screen "performance_1" 1024x761
   IOField "I/O field_73" at 11,174 size 59x47; FormatPattern 99.99
      ProcessValue <- "Suction_press"
   IOField "I/O field_74" at 68,174 size 59x47; FormatPattern 99.99
      ProcessValue <- "Discharge_Press"
   IOField "I/O field_75" at 126,174 size 59x47; FormatPattern 99.99
      ProcessValue <- "Tag_9"
   IOField "I/O field_76" at 185,174 size 59x47; FormatPattern 99.99
      ProcessValue <- "P4"
   IOField "I/O field_77" at 241,174 size 59x47; FormatPattern 99.99
      ProcessValue <- "Torque"
   IOField "I/O field_78" at 299,174 size 59x47; FormatPattern 9999
      ProcessValue <- "RPM"
   IOField "I/O field_79" at 356,174 size 59x47; FormatPattern 99.99
      ProcessValue <- "Tag_33"
   IOField "I/O field_80" at 413,174 size 59x47; FormatPattern 99.99
      ProcessValue <- "VS"
   IOField "I/O field_81" at 470,174 size 59x47; FormatPattern 99.99
      ProcessValue <- "Vd"
   IOField "I/O field_82" at 527,174 size 59x47; FormatPattern 99.99
      ProcessValue <- "Q"
   IOField "I/O field_83" at 586,171 size 59x47; FormatPattern 99.99
      ProcessValue <- "H"
   IOField "I/O field_84" at 642,174 size 59x47; FormatPattern 9999.99
      ProcessValue <- "Shaft_power"
   IOField "I/O field_1" at 700,175 size 59x47; FormatPattern 99.99
      ProcessValue <- "QARS"
   IOField "I/O field_2" at 756,176 size 59x47; FormatPattern 99.99
      ProcessValue <- "H_ARS"
   IOField "I/O field_3" at 813,176 size 59x47; FormatPattern 9999.9
      ProcessValue <- "SP_ARS"
   IOField "I/O field_4" at 870,176 size 59x47; FormatPattern 99.99
      ProcessValue <- "Efficiency"
   IOField "I/O field_5" at 927,178 size 59x47; FormatPattern 99.9
      ProcessValue <- "Npsh"
   IOField "I/O field_6" at 11,220 size 59x47; FormatPattern 99.99
      ProcessValue <- "P1P2_Pressurep1p2{0}"
   IOField "I/O field_7" at 68,220 size 59x47; FormatPattern 99.99
      ProcessValue <- "P1P2_Pressurep1p2{6}"
   IOField "I/O field_8" at 126,220 size 59x47; FormatPattern 99.99
      ProcessValue <- "P3P4_Pressure34{0}"
   IOField "I/O field_9" at 185,220 size 59x47; FormatPattern 99.99
      ProcessValue <- "P3P4_Pressure34{6}"
   IOField "I/O field_10" at 241,220 size 59x47; FormatPattern 99.99
      ProcessValue <- "TS_TS{0}"
   IOField "I/O field_11" at 298,220 size 59x47; FormatPattern 9999
      ProcessValue <- "TS_TS{6}"
   IOField "I/O field_12" at 355,220 size 59x47; FormatPattern 99.99
      ProcessValue <- "Vib_vibration{0}"
   IOField "I/O field_13" at 412,220 size 59x47; FormatPattern 99.99
      ProcessValue <- "VSVD_VsVd{0}"
   IOField "I/O field_14" at 469,220 size 59x47; FormatPattern 99.99
      ProcessValue <- "VSVD_VsVd{6}"
   IOField "I/O field_15" at 527,220 size 59x47; FormatPattern 99.99
      ProcessValue <- "QH_QH{0}"
   IOField "I/O field_16" at 584,220 size 59x47; FormatPattern 99.99
      ProcessValue <- "QH_QH{6}"
   IOField "I/O field_17" at 642,220 size 59x47; FormatPattern 9999.99
      ProcessValue <- "shftP.Pars_shaftP{0}"
   IOField "I/O field_18" at 700,221 size 59x47; FormatPattern 99.99
      ProcessValue <- "QarsHars_QarsHars{0}"
   IOField "I/O field_19" at 756,222 size 59x47; FormatPattern 99.99
      ProcessValue <- "QarsHars_QarsHars{6}"
   IOField "I/O field_20" at 813,223 size 59x47; FormatPattern 9999.99
      ProcessValue <- "shftP.Pars_shaftP{6}"
   IOField "I/O field_21" at 869,224 size 59x47; FormatPattern 99.99
      ProcessValue <- "EFF.NPSH_EFF.NPSH{0}"
   IOField "I/O field_22" at 927,224 size 59x47; FormatPattern 99.99
      ProcessValue <- "EFF.NPSH_EFF.NPSH{6}"
   IOField "I/O field_23" at 11,267 size 59x47; FormatPattern 99.99
      ProcessValue <- "P1P2_Pressurep1p2{1}"
   IOField "I/O field_24" at 68,267 size 59x47; FormatPattern 99.99
      ProcessValue <- "P1P2_Pressurep1p2{7}"
   IOField "I/O field_25" at 126,267 size 59x47; FormatPattern 99.99
      ProcessValue <- "P3P4_Pressure34{1}"
   IOField "I/O field_26" at 185,267 size 59x47; FormatPattern 99.99
      ProcessValue <- "P3P4_Pressure34{7}"
   IOField "I/O field_27" at 241,267 size 59x47; FormatPattern 99.99
      ProcessValue <- "TS_TS{1}"
   IOField "I/O field_28" at 298,267 size 59x47; FormatPattern 9999
      ProcessValue <- "TS_TS{7}"
   IOField "I/O field_29" at 355,267 size 59x47; FormatPattern 99.99
      ProcessValue <- "Vib_vibration{1}"
   IOField "I/O field_30" at 412,267 size 59x47; FormatPattern 99.99
      ProcessValue <- "VSVD_VsVd{1}"
   IOField "I/O field_31" at 469,267 size 59x47; FormatPattern 99.99
      ProcessValue <- "VSVD_VsVd{7}"
   IOField "I/O field_32" at 527,267 size 59x47; FormatPattern 99.99
      ProcessValue <- "QH_QH{1}"
   IOField "I/O field_33" at 584,267 size 59x47; FormatPattern 99.99
      ProcessValue <- "QH_QH{7}"
   IOField "I/O field_34" at 642,267 size 59x47; FormatPattern 9999.99
      ProcessValue <- "shftP.Pars_shaftP{1}"
   IOField "I/O field_35" at 700,267 size 59x47; FormatPattern 99.99
      ProcessValue <- "QarsHars_QarsHars{1}"
   IOField "I/O field_36" at 756,268 size 59x47; FormatPattern 99.99
      ProcessValue <- "QarsHars_QarsHars{7}"
   IOField "I/O field_37" at 813,269 size 59x47; FormatPattern 9999.99
      ProcessValue <- "shftP.Pars_shaftP{7}"
   IOField "I/O field_38" at 869,270 size 59x47; FormatPattern 99.99
      ProcessValue <- "EFF.NPSH_EFF.NPSH{1}"
   IOField "I/O field_39" at 927,270 size 59x47; FormatPattern 99.99
      ProcessValue <- "EFF.NPSH_EFF.NPSH{7}"
   IOField "I/O field_40" at 11,313 size 59x47; FormatPattern 99.99
      ProcessValue <- "P1P2_Pressurep1p2{2}"
   IOField "I/O field_41" at 68,313 size 59x47; FormatPattern 99.99
      ProcessValue <- "P1P2_Pressurep1p2{8}"
   IOField "I/O field_42" at 125,313 size 59x47; FormatPattern 99.99
      ProcessValue <- "P3P4_Pressure34{2}"
   IOField "I/O field_43" at 185,313 size 59x47; FormatPattern 99.99
      ProcessValue <- "P3P4_Pressure34{8}"
   IOField "I/O field_44" at 241,313 size 59x47; FormatPattern 99.99
      ProcessValue <- "TS_TS{2}"
   IOField "I/O field_45" at 298,313 size 59x47; FormatPattern 9999
      ProcessValue <- "TS_TS{8}"
   IOField "I/O field_46" at 355,313 size 59x47; FormatPattern 99.99
      ProcessValue <- "Vib_vibration{2}"
   IOField "I/O field_47" at 412,313 size 59x47; FormatPattern 99.99
      ProcessValue <- "VSVD_VsVd{2}"
   IOField "I/O field_48" at 469,313 size 59x47; FormatPattern 99.99
      ProcessValue <- "VSVD_VsVd{8}"
   IOField "I/O field_49" at 527,313 size 59x47; FormatPattern 99.99
      ProcessValue <- "QH_QH{2}"
   IOField "I/O field_50" at 584,313 size 59x47; FormatPattern 99.99
      ProcessValue <- "QH_QH{8}"
   IOField "I/O field_51" at 642,313 size 59x47; FormatPattern 9999.99
      ProcessValue <- "shftP.Pars_shaftP{2}"
   IOField "I/O field_52" at 700,314 size 59x47; FormatPattern 99.99
      ProcessValue <- "QarsHars_QarsHars{2}"
   IOField "I/O field_53" at 756,314 size 59x47; FormatPattern 99.99
      ProcessValue <- "QarsHars_QarsHars{8}"
   IOField "I/O field_54" at 813,315 size 59x47; FormatPattern 9999.99
      ProcessValue <- "shftP.Pars_shaftP{8}"
   IOField "I/O field_55" at 869,316 size 59x47; FormatPattern 99.99
      ProcessValue <- "EFF.NPSH_EFF.NPSH{2}"
   IOField "I/O field_56" at 927,316 size 59x47; FormatPattern 99.99
      ProcessValue <- "EFF.NPSH_EFF.NPSH{8}"
   IOField "I/O field_57" at 11,359 size 59x47; FormatPattern 99.99
      ProcessValue <- "P1P2_Pressurep1p2{3}"
   IOField "I/O field_58" at 68,359 size 59x47; FormatPattern 99.99
      ProcessValue <- "P1P2_Pressurep1p2{9}"
   IOField "I/O field_59" at 126,359 size 59x47; FormatPattern 99.99
      ProcessValue <- "P3P4_Pressure34{3}"
   IOField "I/O field_60" at 185,359 size 59x47; FormatPattern 99.99
      ProcessValue <- "P3P4_Pressure34{9}"
   IOField "I/O field_61" at 241,359 size 59x47; FormatPattern 99.99
      ProcessValue <- "TS_TS{3}"
   IOField "I/O field_62" at 298,359 size 59x47; FormatPattern 9999
      ProcessValue <- "TS_TS{9}"
   IOField "I/O field_63" at 355,359 size 59x47; FormatPattern 99.99
      ProcessValue <- "Vib_vibration{3}"
   IOField "I/O field_64" at 412,359 size 59x47; FormatPattern 99.99
      ProcessValue <- "VSVD_VsVd{3}"
   IOField "I/O field_65" at 469,359 size 59x47; FormatPattern 99.99
      ProcessValue <- "VSVD_VsVd{9}"
   IOField "I/O field_66" at 527,359 size 59x47; FormatPattern 99.99
      ProcessValue <- "QH_QH{3}"
   IOField "I/O field_67" at 584,359 size 59x47; FormatPattern 99.99
      ProcessValue <- "QH_QH{9}"
   IOField "I/O field_68" at 642,359 size 59x47; FormatPattern 9999.99
      ProcessValue <- "shftP.Pars_shaftP{3}"
   IOField "I/O field_69" at 700,360 size 59x47; FormatPattern 99.99
      ProcessValue <- "QarsHars_QarsHars{3}"
   IOField "I/O field_70" at 756,361 size 59x47; FormatPattern 99.99
      ProcessValue <- "QarsHars_QarsHars{9}"
   IOField "I/O field_71" at 813,361 size 59x47; FormatPattern 9999.99
      ProcessValue <- "shftP.Pars_shaftP{9}"
   IOField "I/O field_72" at 869,363 size 59x47; FormatPattern 99.99
      ProcessValue <- "EFF.NPSH_EFF.NPSH{3}"
   IOField "I/O field_85" at 927,363 size 59x47; FormatPattern 99.99
      ProcessValue <- "EFF.NPSH_EFF.NPSH{9}"
   IOField "I/O field_86" at 10,405 size 59x47; FormatPattern 99.99
      ProcessValue <- "P1P2_Pressurep1p2{4}"
   IOField "I/O field_87" at 68,405 size 59x47; FormatPattern 99.99
      ProcessValue <- "P1P2_Pressurep1p2{10}"
   IOField "I/O field_88" at 126,405 size 59x47; FormatPattern 99.99
      ProcessValue <- "P3P4_Pressure34{4}"
   IOField "I/O field_89" at 185,405 size 59x47; FormatPattern 99.99
      ProcessValue <- "P3P4_Pressure34{10}"
   IOField "I/O field_90" at 241,405 size 59x47; FormatPattern 99.99
      ProcessValue <- "TS_TS{4}"
   IOField "I/O field_91" at 298,405 size 59x47; FormatPattern 9999
      ProcessValue <- "TS_TS{10}"
   IOField "I/O field_92" at 355,405 size 59x47; FormatPattern 99.99
      ProcessValue <- "Vib_vibration{4}"
   IOField "I/O field_93" at 412,405 size 59x47; FormatPattern 99.99
      ProcessValue <- "VSVD_VsVd{4}"
   IOField "I/O field_94" at 469,405 size 59x47; FormatPattern 99.99
      ProcessValue <- "VSVD_VsVd{10}"
   IOField "I/O field_95" at 527,405 size 59x47; FormatPattern 99.99
      ProcessValue <- "QH_QH{4}"
   IOField "I/O field_96" at 584,405 size 59x47; FormatPattern 99.99
      ProcessValue <- "QH_QH{10}"
   IOField "I/O field_97" at 642,405 size 59x47; FormatPattern 9999.99
      ProcessValue <- "shftP.Pars_shaftP{4}"
   IOField "I/O field_98" at 700,406 size 59x47; FormatPattern 99.99
      ProcessValue <- "QarsHars_QarsHars{4}"
   IOField "I/O field_99" at 756,407 size 59x47; FormatPattern 99.99
      ProcessValue <- "QarsHars_QarsHars{10}"
   IOField "I/O field_100" at 813,407 size 59x47; FormatPattern 9999.99
      ProcessValue <- "shftP.Pars_shaftP{10}"
   IOField "I/O field_101" at 869,409 size 59x47; FormatPattern 99.99
      ProcessValue <- "EFF.NPSH_EFF.NPSH{4}"
   IOField "I/O field_102" at 927,409 size 59x47; FormatPattern 99.99
      ProcessValue <- "EFF.NPSH_EFF.NPSH{10}"
   IOField "I/O field_103" at 11,452 size 59x47; FormatPattern 99.99
      ProcessValue <- "P1P2_Pressurep1p2{5}"
   IOField "I/O field_104" at 68,452 size 59x47; FormatPattern 99.99
      ProcessValue <- "P1P2_Pressurep1p2{11}"
   IOField "I/O field_105" at 126,452 size 59x47; FormatPattern 99.99
      ProcessValue <- "P3P4_Pressure34{5}"
   IOField "I/O field_106" at 185,452 size 59x47; FormatPattern 99.99
      ProcessValue <- "P3P4_Pressure34{11}"
   IOField "I/O field_107" at 241,452 size 59x47; FormatPattern 99.99
      ProcessValue <- "TS_TS{5}"
   IOField "I/O field_108" at 298,452 size 59x47; FormatPattern 9999
      ProcessValue <- "TS_TS{11}"
   IOField "I/O field_109" at 355,452 size 59x47; FormatPattern 99.99
      ProcessValue <- "Vib_vibration{5}"
   IOField "I/O field_110" at 412,452 size 59x47; FormatPattern 99.99
      ProcessValue <- "VSVD_VsVd{5}"
   IOField "I/O field_111" at 469,452 size 59x47; FormatPattern 99.99
      ProcessValue <- "VSVD_VsVd{11}"
   IOField "I/O field_112" at 527,452 size 59x47; FormatPattern 99.99
      ProcessValue <- "QH_QH{5}"
   IOField "I/O field_113" at 584,452 size 59x47; FormatPattern 99.99
      ProcessValue <- "QH_QH{11}"
   IOField "I/O field_114" at 642,452 size 59x47; FormatPattern 9999.99
      ProcessValue <- "shftP.Pars_shaftP{5}"
   IOField "I/O field_115" at 700,452 size 59x47; FormatPattern 99.99
      ProcessValue <- "QarsHars_QarsHars{5}"
   IOField "I/O field_116" at 756,453 size 59x47; FormatPattern 99.99
      ProcessValue <- "QarsHars_QarsHars{11}"
   IOField "I/O field_117" at 813,454 size 59x47; FormatPattern 9999.99
      ProcessValue <- "shftP.Pars_shaftP{11}"
   IOField "I/O field_118" at 869,455 size 59x47; FormatPattern 99.99
      ProcessValue <- "EFF.NPSH_EFF.NPSH{5}"
   IOField "I/O field_119" at 927,455 size 59x47; FormatPattern 99.99
      ProcessValue <- "EFF.NPSH_EFF.NPSH{11}"
   Button "Button_2" at 882,555 size 78x51; TextOn 'Rec'; TextOff 'Rec'
      on Press: function_b14e0dd5("record", 0); "linking_to_excel"()
      Appearance <- "record"
   Button "Button_4" at 742,555 size 66x51; TextOff 'up'; PictureOff "Down_Arrow"
      on Press: function_b14e0dd5("Count_up", 0)
   Button "Button_5" at 808,555 size 66x51; TextOff 'down'; PictureOff "Up_Arrow"
      on Press: function_b14e0dd5("count_down", 0)
   Circle "Circle_1" at 997,235 size 16x16
      Appearance <- "Raw1"
   Circle "Circle_2" at 997,281 size 16x16
      Appearance <- "raw2"
   Circle "Circle_3" at 997,326 size 16x16
      Appearance <- "raw3"
   Circle "Circle_4" at 997,374 size 16x16
      Appearance <- "raw4"
   Circle "Circle_5" at 997,421 size 16x16
      Appearance <- "raw5"
   Circle "Circle_6" at 997,465 size 16x16
      Appearance <- "raw6"
   TextField "Text field_1" at 34,132 size 25x23; Text 'P1'
   TextField "Text field_2" at 86,133 size 25x23; Text 'P2'
   TextField "Text field_3" at 143,133 size 25x23; Text 'P3'
   TextField "Text field_4" at 197,133 size 25x23; Text 'P4'
   TextField "Text field_5" at 253,133 size 34x23; Text 'T'
   TextField "Text field_6" at 311,152 size 41x23; Text 'RPM'
   TextField "Text field_7" at 34,156 size 22x23; Text 'bar'
   TextField "Text field_8" at 88,152 size 22x23; Text 'bar'
   TextField "Text field_9" at 144,152 size 22x23; Text 'bar'
   TextField "Text field_10" at 199,152 size 22x23; Text 'bar'
   TextField "Text field_11" at 256,152 size 34x23; Text 'N.m'
   TextField "Text field_12" at 367,129 size 45x23; Text 'Vib.'
   TextField "Text field_13" at 365,153 size 46x23; Text 'mm/s'
   TextField "Text field_14" at 305,131 size 51x20; Text 'speed'
   TextField "Text field_15" at 539,129 size 38x23; Text 'Q'
   TextField "Text field_16" at 542,152 size 42x23; Text 'm3/h'
   TextField "Text field_17" at 595,133 size 33x23; Text 'H'
   TextField "Text field_18" at 601,154 size 24x23; Text 'm'
   TextField "Text field_19" at 636,128 size 63x29; Text 'Shaft p.'
   TextField "Text field_20" at 654,151 size 27x23; Text 'W'
   TextField "Text field_21" at 429,130 size 37x23; Text 'V. s'
   TextField "Text field_22" at 430,152 size 38x23; Text 'm/s'
   TextField "Text field_23" at 483,133 size 35x20; Text 'V. d'
   TextField "Text field_24" at 484,154 size 32x23; Text 'm/s'
   TextField "Text field_25" at 926,133 size 49x23; Text 'NPSH'
   TextField "Text field_26" at 875,133 size 42x23; Text 'Eff.'
   TextField "Text field_27" at 819,133 size 52x20; Text 'P.ref'
   TextField "Text field_28" at 827,157 size 27x23; Text 'W'
   TextField "Text field_29" at 700,133 size 58x23; Text 'Q ref'
   TextField "Text field_30" at 710,154 size 43x23; Text 'm3/h'
   TextField "Text field_31" at 757,133 size 54x23; Text 'H ref'
   TextField "Text field_32" at 770,154 size 27x23; Text 'm'
   Button "Button_10" at 22,697 size 169x56; TextOn 'Home'; TextOff 'Home'
      on Press: ActivateScreen("home", 0)
   Button "Button_11" at 221,695 size 216x57; TextOff 'performance_2'
      on Press: ActivateScreen("performance_2", 0)
   Button "Button_1" at 831,695 size 166x57; TextOn 'Rec'; TextOff 'Cleare All'
      on Press: function_b14e0dd5("clear All", 0)
      Appearance <- "clear All"
   TextField "Text field_37" at 883,153 size 27x23; Text '%'
   TextField "Text field_38" at 939,153 size 27x23; Text 'm'
   Button "Button_3" at 452,695 size 180x57; TextOff 'Trends'
      on Press: ActivateScreen("trends", 0)
   Button "Button_6" at 648,696 size 156x56; TextOn 'Home'; TextOff 'NPSH test'
      on Press: ActivateScreen("NPSH test", 0)
   IOField "I/O field_120" at 390,16 size 105x32; FormatPattern 99999999999999999999
      ProcessValue <- "date"
   IOField "I/O field_121" at 612,14 size 107x32; FormatPattern s9999999999
      ProcessValue <- "time"
   TextField "Text field_33" at 40,14 size 157x38; Text 'Impeller configuration'
   TextField "Text field_34" at 526,11 size 81x38; Text 'Start Time'
   TextField "Text field_35" at 334,16 size 66x38; Text 'Date'
   IOField "I/O field_122" at 836,14 size 107x33; FormatPattern s9999999999
      ProcessValue <- "time_1"
   TextField "Text field_36" at 746,9 size 74x38; Text 'End Time'
   IOField "I/O field_123" at 209,18 size 106x31; FormatPattern ?????????
      ProcessValue <- "configuration"

screen "performance_2" 1024x761
   IOField "I/O field_73" at 11,176 size 59x47; FormatPattern 99.99
      ProcessValue <- "Suction_press"
   IOField "I/O field_74" at 68,174 size 59x47; FormatPattern 99.99
      ProcessValue <- "Discharge_Press"
   IOField "I/O field_75" at 126,174 size 59x47; FormatPattern 99.99
      ProcessValue <- "Tag_9"
   IOField "I/O field_76" at 185,174 size 59x47; FormatPattern 99.99
      ProcessValue <- "P4"
   IOField "I/O field_77" at 241,174 size 59x47; FormatPattern 99.99
      ProcessValue <- "Torque"
   IOField "I/O field_78" at 299,174 size 59x47; FormatPattern 9999
      ProcessValue <- "RPM"
   IOField "I/O field_79" at 356,174 size 59x47; FormatPattern 99.99
      ProcessValue <- "Tag_33"
   IOField "I/O field_80" at 413,174 size 59x47; FormatPattern 99.99
      ProcessValue <- "VS"
   IOField "I/O field_81" at 470,174 size 59x47; FormatPattern 99.99
      ProcessValue <- "Vd"
   IOField "I/O field_82" at 527,174 size 59x47; FormatPattern 99.99
      ProcessValue <- "Q"
   IOField "I/O field_83" at 584,174 size 59x47; FormatPattern 99.99
      ProcessValue <- "H"
   IOField "I/O field_84" at 642,174 size 59x47; FormatPattern 9999.99
      ProcessValue <- "Shaft_power"
   IOField "I/O field_1" at 700,175 size 59x47; FormatPattern 99.99
      ProcessValue <- "QARS"
   IOField "I/O field_2" at 756,176 size 59x47; FormatPattern 99.99
      ProcessValue <- "H_ARS"
   IOField "I/O field_3" at 813,176 size 59x47; FormatPattern 9999.9
      ProcessValue <- "SP_ARS"
   IOField "I/O field_4" at 870,176 size 59x47; FormatPattern 99.99
      ProcessValue <- "Efficiency"
   IOField "I/O field_5" at 927,178 size 59x47; FormatPattern 99.9
      ProcessValue <- "Npsh"
   IOField "I/O field_6" at 11,220 size 59x47; FormatPattern 99.99
      ProcessValue <- "P1P2_Pressurep1p2{0}(1)"
   IOField "I/O field_7" at 68,220 size 59x47; FormatPattern 99.99
      ProcessValue <- "P1P2_Pressurep1p2{0}(7)"
   IOField "I/O field_8" at 126,220 size 59x47; FormatPattern 99.99
      ProcessValue <- "P3P4_Pressure34{0}(1)"
   IOField "I/O field_9" at 185,220 size 59x47; FormatPattern 99.99
      ProcessValue <- "P3P4_Pressure34{6}(1)"
   IOField "I/O field_10" at 241,220 size 59x47; FormatPattern 99.99
      ProcessValue <- "TS_TS{0}(1)"
   IOField "I/O field_11" at 298,220 size 59x47; FormatPattern 9999
      ProcessValue <- "TS_TS{6}(1)"
   IOField "I/O field_12" at 355,220 size 59x47; FormatPattern 99.99
      ProcessValue <- "Vib_vibration{0}(1)"
   IOField "I/O field_13" at 412,220 size 59x47; FormatPattern 99.99
      ProcessValue <- "VSVD_VsVd{0}(1)"
   IOField "I/O field_14" at 469,220 size 59x47; FormatPattern 99.99
      ProcessValue <- "VSVD_VsVd{6}(1)"
   IOField "I/O field_15" at 527,220 size 59x47; FormatPattern 99.99
      ProcessValue <- "QH_QH{0}(1)"
   IOField "I/O field_16" at 584,220 size 59x47; FormatPattern 99.99
      ProcessValue <- "QH_QH{6}(1)"
   IOField "I/O field_17" at 642,220 size 59x47; FormatPattern 9999.99
      ProcessValue <- "shftP.Pars_shaftP{0}(1)"
   IOField "I/O field_18" at 700,221 size 59x47; FormatPattern 99.99
      ProcessValue <- "QarsHars_QarsHars{0}(1)"
   IOField "I/O field_19" at 756,222 size 59x47; FormatPattern 99.99
      ProcessValue <- "QarsHars_QarsHars{6}(1)"
   IOField "I/O field_20" at 813,223 size 59x47; FormatPattern 9999.99
      ProcessValue <- "shftP.Pars_shaftP{6}(1)"
   IOField "I/O field_21" at 869,224 size 59x47; FormatPattern 99.99
      ProcessValue <- "EFF.NPSH_EFF.NPSH{0}(1)"
   IOField "I/O field_22" at 927,224 size 59x47; FormatPattern 99.99
      ProcessValue <- "EFF.NPSH_EFF.NPSH{6}(1)"
   IOField "I/O field_23" at 11,267 size 59x47; FormatPattern 99.99
      ProcessValue <- "P1P2_Pressurep1p2{0}(2)"
   IOField "I/O field_24" at 68,267 size 59x47; FormatPattern 99.99
      ProcessValue <- "P1P2_Pressurep1p2{0}(8)"
   IOField "I/O field_25" at 126,267 size 59x47; FormatPattern 99.99
      ProcessValue <- "P3P4_Pressure34{1}(1)"
   IOField "I/O field_26" at 185,267 size 59x47; FormatPattern 99.99
      ProcessValue <- "P3P4_Pressure34{7}(1)"
   IOField "I/O field_27" at 241,267 size 59x47; FormatPattern 99.99
      ProcessValue <- "TS_TS{1}(1)"
   IOField "I/O field_28" at 298,267 size 59x47; FormatPattern 9999
      ProcessValue <- "TS_TS{7}(1)"
   IOField "I/O field_29" at 355,267 size 59x47; FormatPattern 99.99
      ProcessValue <- "Vib_vibration{1}(1)"
   IOField "I/O field_30" at 412,267 size 59x47; FormatPattern 99.99
      ProcessValue <- "VSVD_VsVd{1}(1)"
   IOField "I/O field_31" at 469,267 size 59x47; FormatPattern 99.99
      ProcessValue <- "VSVD_VsVd{7}(1)"
   IOField "I/O field_32" at 527,267 size 59x47; FormatPattern 99.99
      ProcessValue <- "QH_QH{1}(1)"
   IOField "I/O field_33" at 584,267 size 59x47; FormatPattern 99.99
      ProcessValue <- "QH_QH{7}(1)"
   IOField "I/O field_34" at 642,267 size 59x47; FormatPattern 9999.99
      ProcessValue <- "shftP.Pars_shaftP{1}(1)"
   IOField "I/O field_35" at 700,267 size 59x47; FormatPattern 99.99
      ProcessValue <- "QarsHars_QarsHars{1}(1)"
   IOField "I/O field_36" at 756,268 size 59x47; FormatPattern 99.99
      ProcessValue <- "QarsHars_QarsHars{7}(1)"
   IOField "I/O field_37" at 813,269 size 59x47; FormatPattern 9999.99
      ProcessValue <- "shftP.Pars_shaftP{7}(1)"
   IOField "I/O field_38" at 869,270 size 59x47; FormatPattern 99.99
      ProcessValue <- "EFF.NPSH_EFF.NPSH{1}(1)"
   IOField "I/O field_39" at 927,270 size 59x47; FormatPattern 99.99
      ProcessValue <- "EFF.NPSH_EFF.NPSH{7}(1)"
   IOField "I/O field_40" at 11,313 size 59x47; FormatPattern 99.99
      ProcessValue <- "P1P2_Pressurep1p2{0}(3)"
   IOField "I/O field_41" at 68,313 size 59x47; FormatPattern 99.99
      ProcessValue <- "P1P2_Pressurep1p2{0}(9)"
   IOField "I/O field_42" at 125,313 size 59x47; FormatPattern 99.99
      ProcessValue <- "P3P4_Pressure34{2}(1)"
   IOField "I/O field_43" at 185,313 size 59x47; FormatPattern 99.99
      ProcessValue <- "P3P4_Pressure34{8}(1)"
   IOField "I/O field_44" at 241,313 size 59x47; FormatPattern 99.99
      ProcessValue <- "TS_TS{2}(1)"
   IOField "I/O field_45" at 298,313 size 59x47; FormatPattern 9999
      ProcessValue <- "TS_TS{8}(1)"
   IOField "I/O field_46" at 355,313 size 59x47; FormatPattern 99.99
      ProcessValue <- "Vib_vibration{2}(1)"
   IOField "I/O field_47" at 412,313 size 59x47; FormatPattern 99.99
      ProcessValue <- "VSVD_VsVd{2}(1)"
   IOField "I/O field_48" at 469,313 size 59x47; FormatPattern 99.99
      ProcessValue <- "VSVD_VsVd{8}(1)"
   IOField "I/O field_49" at 527,313 size 59x47; FormatPattern 99.99
      ProcessValue <- "QH_QH{2}(1)"
   IOField "I/O field_50" at 584,313 size 59x47; FormatPattern 99.99
      ProcessValue <- "QH_QH{8}(1)"
   IOField "I/O field_51" at 642,313 size 59x47; FormatPattern 9999.99
      ProcessValue <- "shftP.Pars_shaftP{2}(1)"
   IOField "I/O field_52" at 700,314 size 59x47; FormatPattern 99.99
      ProcessValue <- "QarsHars_QarsHars{2}(1)"
   IOField "I/O field_53" at 756,314 size 59x47; FormatPattern 99.99
      ProcessValue <- "QarsHars_QarsHars{8}(1)"
   IOField "I/O field_54" at 813,315 size 59x47; FormatPattern 9999.99
      ProcessValue <- "shftP.Pars_shaftP{8}(1)"
   IOField "I/O field_55" at 869,316 size 59x47; FormatPattern 99.99
      ProcessValue <- "EFF.NPSH_EFF.NPSH{2}(1)"
   IOField "I/O field_56" at 927,316 size 59x47; FormatPattern 99.99
      ProcessValue <- "EFF.NPSH_EFF.NPSH{8}(1)"
   IOField "I/O field_57" at 11,359 size 59x47; FormatPattern 99.99
      ProcessValue <- "P1P2_Pressurep1p2{0}(4)"
   IOField "I/O field_58" at 68,359 size 59x47; FormatPattern 99.99
      ProcessValue <- "P1P2_Pressurep1p2{0}(10)"
   IOField "I/O field_59" at 126,359 size 59x47; FormatPattern 99.99
      ProcessValue <- "P3P4_Pressure34{3}(1)"
   IOField "I/O field_60" at 185,359 size 59x47; FormatPattern 99.99
      ProcessValue <- "P3P4_Pressure34{9}(1)"
   IOField "I/O field_61" at 241,359 size 59x47; FormatPattern 99.99
      ProcessValue <- "TS_TS{3}(1)"
   IOField "I/O field_62" at 298,359 size 59x47; FormatPattern 9999
      ProcessValue <- "TS_TS{9}(1)"
   IOField "I/O field_63" at 355,359 size 59x47; FormatPattern 99.99
      ProcessValue <- "Vib_vibration{3}(1)"
   IOField "I/O field_64" at 412,359 size 59x47; FormatPattern 99.99
      ProcessValue <- "VSVD_VsVd{3}(1)"
   IOField "I/O field_65" at 469,359 size 59x47; FormatPattern 99.99
      ProcessValue <- "VSVD_VsVd{9}(1)"
   IOField "I/O field_66" at 527,359 size 59x47; FormatPattern 99.99
      ProcessValue <- "QH_QH{3}(1)"
   IOField "I/O field_67" at 584,359 size 59x47; FormatPattern 99.99
      ProcessValue <- "QH_QH{9}(1)"
   IOField "I/O field_68" at 642,359 size 59x47; FormatPattern 9999.99
      ProcessValue <- "shftP.Pars_shaftP{3}(1)"
   IOField "I/O field_69" at 700,360 size 59x47; FormatPattern 99.99
      ProcessValue <- "QarsHars_QarsHars{3}(1)"
   IOField "I/O field_70" at 756,361 size 59x47; FormatPattern 99.99
      ProcessValue <- "QarsHars_QarsHars{9}(1)"
   IOField "I/O field_71" at 813,361 size 59x47; FormatPattern 9999.99
      ProcessValue <- "shftP.Pars_shaftP{9}(1)"
   IOField "I/O field_72" at 869,363 size 59x47; FormatPattern 99.99
      ProcessValue <- "EFF.NPSH_EFF.NPSH{3}(1)"
   IOField "I/O field_85" at 927,363 size 59x47; FormatPattern 99.99
      ProcessValue <- "EFF.NPSH_EFF.NPSH{9}(1)"
   IOField "I/O field_86" at 10,405 size 59x47; FormatPattern 99.99
      ProcessValue <- "P1P2_Pressurep1p2{0}(5)"
   IOField "I/O field_87" at 68,405 size 59x47; FormatPattern 99.99
      ProcessValue <- "P1P2_Pressurep1p2{0}(11)"
   IOField "I/O field_88" at 126,405 size 59x47; FormatPattern 99.99
      ProcessValue <- "P3P4_Pressure34{4}(1)"
   IOField "I/O field_89" at 185,405 size 59x47; FormatPattern 99.99
      ProcessValue <- "P3P4_Pressure34{10}(1)"
   IOField "I/O field_90" at 241,405 size 59x47; FormatPattern 99.99
      ProcessValue <- "TS_TS{4}(1)"
   IOField "I/O field_91" at 298,405 size 59x47; FormatPattern 9999
      ProcessValue <- "TS_TS{10}(1)"
   IOField "I/O field_92" at 355,405 size 59x47; FormatPattern 99.99
      ProcessValue <- "Vib_vibration{4}(1)"
   IOField "I/O field_93" at 412,405 size 59x47; FormatPattern 99.99
      ProcessValue <- "VSVD_VsVd{4}(1)"
   IOField "I/O field_94" at 469,405 size 59x47; FormatPattern 99.99
      ProcessValue <- "VSVD_VsVd{10}(1)"
   IOField "I/O field_95" at 527,405 size 59x47; FormatPattern 99.99
      ProcessValue <- "QH_QH{4}(1)"
   IOField "I/O field_96" at 584,405 size 59x47; FormatPattern 99.99
      ProcessValue <- "QH_QH{10}(1)"
   IOField "I/O field_97" at 642,405 size 59x47; FormatPattern 9999.99
      ProcessValue <- "shftP.Pars_shaftP{4}(1)"
   IOField "I/O field_98" at 700,406 size 59x47; FormatPattern 99.99
      ProcessValue <- "QarsHars_QarsHars{4}(1)"
   IOField "I/O field_99" at 756,407 size 59x47; FormatPattern 99.99
      ProcessValue <- "QarsHars_QarsHars{10}(1)"
   IOField "I/O field_100" at 813,407 size 59x47; FormatPattern 9999.99
      ProcessValue <- "shftP.Pars_shaftP{10}(1)"
   IOField "I/O field_101" at 869,409 size 59x47; FormatPattern 99.99
      ProcessValue <- "EFF.NPSH_EFF.NPSH{4}(1)"
   IOField "I/O field_102" at 927,409 size 59x47; FormatPattern 99.99
      ProcessValue <- "EFF.NPSH_EFF.NPSH{10}(1)"
   IOField "I/O field_103" at 11,452 size 59x47; FormatPattern 99.99
      ProcessValue <- "P1P2_Pressurep1p2{0}(6)"
   IOField "I/O field_104" at 68,452 size 59x47; FormatPattern 99.99
      ProcessValue <- "P1P2_Pressurep1p2{0}(12)"
   IOField "I/O field_105" at 126,452 size 59x47; FormatPattern 99.99
      ProcessValue <- "P3P4_Pressure34{5}(1)"
   IOField "I/O field_106" at 185,452 size 59x47; FormatPattern 99.99
      ProcessValue <- "P3P4_Pressure34{11}(1)"
   IOField "I/O field_107" at 241,452 size 59x47; FormatPattern 99.99
      ProcessValue <- "TS_TS{5}(1)"
   IOField "I/O field_108" at 298,452 size 59x47; FormatPattern 9999
      ProcessValue <- "TS_TS{11}(1)"
   IOField "I/O field_109" at 355,452 size 59x47; FormatPattern 99.99
      ProcessValue <- "Vib_vibration{5}(1)"
   IOField "I/O field_110" at 412,452 size 59x47; FormatPattern 99.99
      ProcessValue <- "VSVD_VsVd{5}(1)"
   IOField "I/O field_111" at 469,452 size 59x47; FormatPattern 99.99
      ProcessValue <- "VSVD_VsVd{11}(1)"
   IOField "I/O field_112" at 527,452 size 59x47; FormatPattern 99.99
      ProcessValue <- "QH_QH{5}(1)"
   IOField "I/O field_113" at 584,452 size 59x47; FormatPattern 99.99
      ProcessValue <- "QH_QH{11}(1)"
   IOField "I/O field_114" at 642,452 size 59x47; FormatPattern 9999.99
      ProcessValue <- "shftP.Pars_shaftP{5}(1)"
   IOField "I/O field_115" at 700,452 size 59x47; FormatPattern 99.99
      ProcessValue <- "QarsHars_QarsHars{5}(1)"
   IOField "I/O field_116" at 756,453 size 59x47; FormatPattern 99.99
      ProcessValue <- "QarsHars_QarsHars{11}(1)"
   IOField "I/O field_117" at 813,454 size 59x47; FormatPattern 9999.99
      ProcessValue <- "shftP.Pars_shaftP{11}(1)"
   IOField "I/O field_118" at 869,455 size 59x47; FormatPattern 99.99
      ProcessValue <- "EFF.NPSH_EFF.NPSH{5}(1)"
   IOField "I/O field_119" at 927,455 size 59x47; FormatPattern 99.99
      ProcessValue <- "EFF.NPSH_EFF.NPSH{11}(1)"
   Button "Button_2" at 882,555 size 78x51; TextOn 'Rec'; TextOff 'Rec'
      on Press: function_b14e0dd5("record", 0); "linking_to_excel"()
      Appearance <- "record"
   Button "Button_4" at 742,555 size 66x51; TextOff 'up'; PictureOff "Down_Arrow"
      on Press: function_b14e0dd5("Count_up", 0)
   Button "Button_5" at 808,555 size 66x51; TextOff 'down'; PictureOff "Up_Arrow"
      on Press: function_b14e0dd5("count_down", 0)
   Circle "Circle_1" at 997,235 size 16x16
      Appearance <- "raw7"
   Circle "Circle_2" at 997,281 size 16x16
      Appearance <- "raw8"
   Circle "Circle_3" at 997,326 size 16x16
      Appearance <- "raw9"
   Circle "Circle_4" at 997,374 size 16x16
      Appearance <- "raw10"
   Circle "Circle_5" at 997,421 size 16x16
      Appearance <- "raw11"
   Circle "Circle_6" at 997,465 size 16x16
      Appearance <- "raw12"
   TextField "Text field_1" at 34,132 size 25x23; Text 'P1'
   TextField "Text field_2" at 86,133 size 25x23; Text 'P2'
   TextField "Text field_3" at 143,133 size 25x23; Text 'P3'
   TextField "Text field_4" at 197,133 size 25x23; Text 'P4'
   TextField "Text field_5" at 253,133 size 34x23; Text 'T'
   TextField "Text field_6" at 311,152 size 41x23; Text 'RPM'
   TextField "Text field_7" at 34,156 size 22x23; Text 'bar'
   TextField "Text field_8" at 88,152 size 22x23; Text 'bar'
   TextField "Text field_9" at 144,152 size 22x23; Text 'bar'
   TextField "Text field_10" at 199,152 size 22x23; Text 'bar'
   TextField "Text field_11" at 256,152 size 34x23; Text 'N.m'
   TextField "Text field_12" at 367,129 size 45x23; Text 'Vib.'
   TextField "Text field_13" at 365,153 size 46x23; Text 'mm/s'
   TextField "Text field_14" at 305,131 size 51x20; Text 'speed'
   TextField "Text field_15" at 539,129 size 38x23; Text 'Q'
   TextField "Text field_16" at 542,152 size 42x23; Text 'm3/h'
   TextField "Text field_17" at 595,133 size 33x23; Text 'H'
   TextField "Text field_18" at 601,154 size 24x23; Text 'm'
   TextField "Text field_19" at 636,128 size 63x29; Text 'Shaft p.'
   TextField "Text field_20" at 654,151 size 27x23; Text 'W'
   TextField "Text field_21" at 429,130 size 37x23; Text 'V. s'
   TextField "Text field_22" at 430,152 size 38x23; Text 'm/s'
   TextField "Text field_23" at 483,133 size 35x20; Text 'V. d'
   TextField "Text field_24" at 484,154 size 32x23; Text 'm/s'
   TextField "Text field_25" at 926,133 size 49x23; Text 'NPSH'
   TextField "Text field_26" at 875,133 size 42x23; Text 'Eff.'
   TextField "Text field_27" at 819,133 size 52x20; Text 'P.ref'
   TextField "Text field_28" at 828,154 size 27x23; Text 'W'
   TextField "Text field_29" at 700,133 size 58x23; Text 'Q ref'
   TextField "Text field_30" at 710,154 size 43x23; Text 'm3/h'
   TextField "Text field_31" at 757,133 size 54x23; Text 'H ref'
   TextField "Text field_32" at 770,154 size 27x23; Text 'm'
   Button "Button_10" at 23,697 size 169x56; TextOn 'Home'; TextOff 'Home'
      on Press: ActivateScreen("home", 0)
   Button "Button_11" at 214,695 size 196x57; TextOff 'performance_1'
      on Press: ActivateScreen("performance_1", 0)
   Button "Button_1" at 827,695 size 153x57; TextOn 'Rec'; TextOff 'Cleare All'
      on Press: function_b14e0dd5("clear All", 0)
      Appearance <- "clear All"
   TextField "Text field_37" at 883,153 size 27x23; Text '%'
   TextField "Text field_38" at 939,153 size 27x23; Text 'm'
   Button "Button_3" at 427,693 size 140x57; TextOff 'Trends'
      on Press: ActivateScreen("trends", 0)
   Button "Button_6" at 612,696 size 156x56; TextOn 'Home'; TextOff 'NPSH test'
      on Press: ActivateScreen("NPSH test", 0)
   IOField "I/O field_120" at 390,16 size 105x32; FormatPattern 99999999999999999999
      ProcessValue <- "date"
   IOField "I/O field_121" at 612,14 size 107x32; FormatPattern s9999999999
      ProcessValue <- "time"
   TextField "Text field_33" at 40,14 size 157x38; Text 'Impeller configuration'
   TextField "Text field_34" at 526,11 size 81x38; Text 'Start Time'
   TextField "Text field_35" at 334,16 size 66x38; Text 'Date'
   IOField "I/O field_122" at 836,14 size 107x33; FormatPattern s9999999999
      ProcessValue <- "time_1"
   TextField "Text field_36" at 746,9 size 74x38; Text 'End Time'
   IOField "I/O field_123" at 209,18 size 106x31; FormatPattern ?????????
      ProcessValue <- "configuration"

screen "trends" 1024x761
   Button "Button_10" at 23,697 size 158x56; TextOn 'Home'; TextOff 'Home'
      on Press: ActivateScreen("home", 0)
   Button "Button_11" at 208,695 size 188x57; TextOff 'performance_1'
      on Press: ActivateScreen("performance_1", 0)
   Button "Button_3" at 429,697 size 199x57; TextOff 'performance_2'
      on Press: ActivateScreen("performance_2", 0)
   Button "Button_2" at 843,693 size 156x56; TextOff 'Exit'
      on Press: StopRuntime(0)
   FunctionTrendControl "f(x) trend view_1" at 234,158 size 775x410
   Button "Button_1" at 651,696 size 156x56; TextOn 'Home'; TextOff 'NPSH test'
      on Press: ActivateScreen("NPSH test", 0)
   IOField "I/O field_8" at 390,16 size 105x32; FormatPattern 99999999999999999999
      ProcessValue <- "date"
   IOField "I/O field_9" at 612,14 size 107x32; FormatPattern s9999999999
      ProcessValue <- "time"
   TextField "Text field_8" at 40,14 size 157x38; Text 'Impeller configuration'
   TextField "Text field_9" at 526,11 size 81x38; Text 'Start Time'
   TextField "Text field_10" at 334,16 size 66x38; Text 'Date'
   IOField "I/O field_10" at 836,14 size 107x33; FormatPattern s9999999999
      ProcessValue <- "time_1"
   TextField "Text field_11" at 746,9 size 74x38; Text 'End Time'
   IOField "I/O field_7" at 209,18 size 106x31; FormatPattern ?????????
      ProcessValue <- "configuration"

screen "NPSH test" 1024x761
   Button "Button_2" at 858,698 size 156x56; TextOff 'Exit'
      on Press: StopRuntime(0)
   IOField "I/O field_73" at 11,174 size 59x47; FormatPattern 99.99
      ProcessValue <- "Suction_press"
   IOField "I/O field_6" at 11,220 size 59x47; FormatPattern 99.99
      ProcessValue <- "P1P2_Pressurep1p2{0}"
   IOField "I/O field_23" at 11,267 size 59x47; FormatPattern 99.99
      ProcessValue <- "P1P2_Pressurep1p2{1}"
   IOField "I/O field_40" at 11,313 size 59x47; FormatPattern 99.99
      ProcessValue <- "P1P2_Pressurep1p2{2}"
   IOField "I/O field_57" at 11,359 size 59x47; FormatPattern 99.99
      ProcessValue <- "P1P2_Pressurep1p2{3}"
   IOField "I/O field_86" at 10,405 size 59x47; FormatPattern 99.99
      ProcessValue <- "P1P2_Pressurep1p2{4}"
   TextField "Text field_1" at 34,132 size 25x23; Text 'P1'
   TextField "Text field_7" at 34,156 size 22x23; Text 'bar'
   IOField "I/O field_82" at 244,174 size 59x47; FormatPattern 99.99
      ProcessValue <- "Q"
   IOField "I/O field_83" at 301,174 size 59x47; FormatPattern 99.99
      ProcessValue <- "H"
   IOField "I/O field_15" at 244,220 size 59x47; FormatPattern 99.99
      ProcessValue <- "QH_QH{0}"
   IOField "I/O field_16" at 301,220 size 59x47; FormatPattern 99.99
      ProcessValue <- "QH_QH{6}"
   IOField "I/O field_32" at 244,267 size 59x47; FormatPattern 99.99
      ProcessValue <- "QH_QH{1}"
   IOField "I/O field_33" at 301,267 size 59x47; FormatPattern 99.99
      ProcessValue <- "QH_QH{7}"
   IOField "I/O field_49" at 244,313 size 59x47; FormatPattern 99.99
      ProcessValue <- "QH_QH{2}"
   IOField "I/O field_50" at 301,313 size 59x47; FormatPattern 99.99
      ProcessValue <- "QH_QH{8}"
   IOField "I/O field_66" at 244,359 size 59x47; FormatPattern 99.99
      ProcessValue <- "QH_QH{3}"
   IOField "I/O field_67" at 301,359 size 59x47; FormatPattern 99.99
      ProcessValue <- "QH_QH{9}"
   IOField "I/O field_95" at 244,405 size 59x47; FormatPattern 99.99
      ProcessValue <- "QH_QH{4}"
   IOField "I/O field_96" at 301,405 size 59x47; FormatPattern 99.99
      ProcessValue <- "QH_QH{10}"
   TextField "Text field_15" at 256,129 size 38x23; Text 'Q'
   TextField "Text field_16" at 259,152 size 42x23; Text 'm3/h'
   TextField "Text field_17" at 312,133 size 33x23; Text 'H'
   TextField "Text field_18" at 318,154 size 24x23; Text 'm'
   IOField "I/O field_5" at 420,175 size 59x47; FormatPattern 99.9
      ProcessValue <- "Npsh"
   IOField "I/O field_22" at 420,221 size 59x47; FormatPattern 99.99
      ProcessValue <- "EFF.NPSH_EFF.NPSH{6}"
   IOField "I/O field_39" at 420,267 size 59x47; FormatPattern 99.99
      ProcessValue <- "EFF.NPSH_EFF.NPSH{7}"
   IOField "I/O field_56" at 420,314 size 59x47; FormatPattern 99.99
      ProcessValue <- "EFF.NPSH_EFF.NPSH{8}"
   IOField "I/O field_85" at 420,360 size 59x47; FormatPattern 99.99
      ProcessValue <- "EFF.NPSH_EFF.NPSH{9}"
   IOField "I/O field_102" at 420,406 size 59x47; FormatPattern 99.99
      ProcessValue <- "EFF.NPSH_EFF.NPSH{10}"
   Circle "Circle_1" at 496,231 size 16x16
      Appearance <- "Raw1"
   Circle "Circle_2" at 496,277 size 16x16
      Appearance <- "raw2"
   Circle "Circle_3" at 496,323 size 16x16
      Appearance <- "raw3"
   Circle "Circle_4" at 496,370 size 16x16
      Appearance <- "raw4"
   Circle "Circle_5" at 496,417 size 16x16
      Appearance <- "raw5"
   TextField "Text field_25" at 418,130 size 49x23; Text 'NPSH'
   TextField "Text field_38" at 431,150 size 27x23; Text 'm'
   IOField "I/O field_1" at 358,174 size 59x47; FormatPattern 99.99
      ProcessValue <- "deviation"
   IOField "I/O field_2" at 358,220 size 59x47; FormatPattern 99.99
      ProcessValue <- "deviation_0"
   IOField "I/O field_3" at 358,267 size 59x47; FormatPattern 99.99
      ProcessValue <- "deviation_1"
   IOField "I/O field_4" at 358,313 size 59x47; FormatPattern 99.99
      ProcessValue <- "deviation_2"
   IOField "I/O field_7" at 358,359 size 59x47; FormatPattern 99.99
      ProcessValue <- "deviation_3"
   IOField "I/O field_8" at 358,405 size 59x47; FormatPattern 99.99
      ProcessValue <- "deviation_4"
   TextField "Text field_2" at 356,129 size 63x23; Text 'deviation'
   TextField "Text field_3" at 369,149 size 27x23; Text '%'
   IOField "I/O field_9" at 10,455 size 59x47; FormatPattern 99.99
      ProcessValue <- "P1P2_Pressurep1p2{5}"
   IOField "I/O field_10" at 243,454 size 59x47; FormatPattern 99.99
      ProcessValue <- "QH_QH{5}"
   IOField "I/O field_11" at 300,455 size 59x47; FormatPattern 99.99
      ProcessValue <- "QH_QH{11}"
   IOField "I/O field_12" at 419,454 size 59x47; FormatPattern 99.99
      ProcessValue <- "EFF.NPSH_EFF.NPSH{11}"
   IOField "I/O field_13" at 357,455 size 59x47; FormatPattern 99.99
      ProcessValue <- "deviation_5"
   IOField "I/O field_74" at 68,174 size 59x47; FormatPattern 99.99
      ProcessValue <- "Discharge_Press"
   IOField "I/O field_75" at 126,174 size 59x47; FormatPattern 99.99
      ProcessValue <- "Tag_9"
   IOField "I/O field_76" at 185,174 size 59x47; FormatPattern 99.99
      ProcessValue <- "P4"
   IOField "I/O field_14" at 68,220 size 59x47; FormatPattern 99.99
      ProcessValue <- "P1P2_Pressurep1p2{6}"
   IOField "I/O field_17" at 126,220 size 59x47; FormatPattern 99.99
      ProcessValue <- "P3P4_Pressure34{0}"
   IOField "I/O field_18" at 185,220 size 59x47; FormatPattern 99.99
      ProcessValue <- "P3P4_Pressure34{6}"
   IOField "I/O field_24" at 68,267 size 59x47; FormatPattern 99.99
      ProcessValue <- "P1P2_Pressurep1p2{7}"
   IOField "I/O field_25" at 126,267 size 59x47; FormatPattern 99.99
      ProcessValue <- "P3P4_Pressure34{1}"
   IOField "I/O field_26" at 185,267 size 59x47; FormatPattern 99.99
      ProcessValue <- "P3P4_Pressure34{7}"
   IOField "I/O field_41" at 68,313 size 59x47; FormatPattern 99.99
      ProcessValue <- "P1P2_Pressurep1p2{8}"
   IOField "I/O field_42" at 125,313 size 59x47; FormatPattern 99.99
      ProcessValue <- "P3P4_Pressure34{2}"
   IOField "I/O field_43" at 185,313 size 59x47; FormatPattern 99.99
      ProcessValue <- "P3P4_Pressure34{8}"
   IOField "I/O field_58" at 68,359 size 59x47; FormatPattern 99.99
      ProcessValue <- "P1P2_Pressurep1p2{9}"
   IOField "I/O field_59" at 126,359 size 59x47; FormatPattern 99.99
      ProcessValue <- "P3P4_Pressure34{3}"
   IOField "I/O field_60" at 185,359 size 59x47; FormatPattern 99.99
      ProcessValue <- "P3P4_Pressure34{9}"
   IOField "I/O field_87" at 68,405 size 59x47; FormatPattern 99.99
      ProcessValue <- "P1P2_Pressurep1p2{10}"
   IOField "I/O field_88" at 126,405 size 59x47; FormatPattern 99.99
      ProcessValue <- "P3P4_Pressure34{4}"
   IOField "I/O field_89" at 185,405 size 59x47; FormatPattern 99.99
      ProcessValue <- "P3P4_Pressure34{10}"
   IOField "I/O field_104" at 68,452 size 59x47; FormatPattern 99.99
      ProcessValue <- "P1P2_Pressurep1p2{11}"
   IOField "I/O field_105" at 126,452 size 59x47; FormatPattern 99.99
      ProcessValue <- "P3P4_Pressure34{5}"
   IOField "I/O field_106" at 185,452 size 59x47; FormatPattern 99.99
      ProcessValue <- "P3P4_Pressure34{11}"
   TextField "Text field_5" at 86,133 size 25x23; Text 'P2'
   TextField "Text field_6" at 143,133 size 25x23; Text 'P3'
   TextField "Text field_8" at 197,133 size 25x23; Text 'P4'
   TextField "Text field_9" at 88,152 size 22x23; Text 'bar'
   TextField "Text field_10" at 144,152 size 22x23; Text 'bar'
   TextField "Text field_11" at 199,152 size 22x23; Text 'bar'
   Button "Button_1" at 439,544 size 78x51; TextOn 'Rec'; TextOff 'Rec'
      on Press: function_b14e0dd5("record", 0); "linking_to_excel"()
      Appearance <- "record"
   Button "Button_4" at 300,545 size 66x51; TextOff 'up'; PictureOff "Down_Arrow"
      on Press: function_b14e0dd5("Count_up", 0)
   Button "Button_5" at 366,544 size 66x51; TextOff 'down'; PictureOff "Up_Arrow"
      on Press: function_b14e0dd5("count_down", 0)
   FunctionTrendControl "f(x) trend view_1" at 526,148 size 494x365
   Button "Button_10" at 23,697 size 169x56; TextOn 'Home'; TextOff 'Home'
      on Press: ActivateScreen("home", 0)
   Button "Button_11" at 207,695 size 189x56; TextOff 'performance_1'
      on Press: ActivateScreen("performance_1", 0)
   Button "Button_3" at 439,697 size 191x56; TextOff 'performance_2'
      on Press: ActivateScreen("performance_2", 0)
   Button "Button_6" at 665,698 size 140x56; TextOff 'Trends'
      on Press: ActivateScreen("trends", 0)
   Button "Button_7" at 416,26 size 102x23; TextOff 'NPSH test'
      on Click: ActivateScreen("NPSH test", 0)
   Button "Button_8" at 800,43 size 51x23; TextOff 'Text'
   Button "Button_9" at 115,75 size 64x36; TextOff 'Open'
      on Press: function_b14e0dd5("stepp1_start", 0)
      Appearance <- "stepp1_start"
   IOField "I/O field_19" at 115,43 size 64x32; FormatPattern 99.9
      ProcessValue <- "stepp1_distance"
   Circle "Circle_6" at 495,466 size 16x16
      Appearance <- "raw6"
   Button "Button_12" at 22,59 size 92x40; TextOff 'Stepp1_Enab.'
      on Press: InvertBit("stepp1_enab")
      Appearance <- "stepp1_enab"
   Button "Button_13" at 209,61 size 94x38; TextOff 'Stepp2_Enab.'
      on Press: InvertBit("stepp2_enab")
      Appearance <- "stepp2_enab"
   IOField "I/O field_20" at 304,47 size 64x32; FormatPattern 99.9
      ProcessValue <- "stepp2_distance"
   Button "Button_14" at 304,80 size 64x36; TextOff 'Open'
      on Press: function_b14e0dd5("stepp2_excut", 0)
      Appearance <- "stepp2_excut"
   IOField "I/O field_21" at 630,94 size 68x32; FormatPattern 999.9; Unit   C
      ProcessValue <- "Temperature"
   TextField "Text field_4" at 598,60 size 129x23; Text 'Water Tempreture'

screen "Temp&Vib_trends" 1024x761
   TrendView "Trend view_1" at 23,68 size 446x459
   TrendView "Trend view_2" at 483,69 size 458x459
   Button "Button_1" at 205,560 size 99x23; TextOff 'Tempreture'
   Button "Button_2" at 667,555 size 96x23; TextOff 'vibration'
   Button "Button_3" at 858,698 size 156x56; TextOff 'Exit'
      on Press: StopRuntime(0)
   Button "Button_10" at 594,699 size 169x56; TextOn 'Home'; TextOff 'Home'
      on Press: ActivateScreen("home", 0)
   Button "Button_4" at 394,16 size 165x36; TextOff 'Temp&Vib_trends'
      on Click: ActivateScreen("Temp&Vib_trends", 0)

VB script "linking_to_excel"
   Dim objExcel, strExcelPath, strSaveAsPath, objSheet
   
   strExcelPath = "C:\Users\DELL\Desktop_Perfomance test impeller Configration STD & D110 & D120 & D130 at all RPM.xlsx"
   strSaveAsPath = "C:\Users\DELL\Desktop\performance.xlsx"
   ' Open specified spreadsheet and select the first worksheet.
   Set objExcel = CreateObject("Excel.Application")
   objExcel.Workbooks.Open strExcelPath
   Set objSheet = objExcel.ActiveWorkbook.Worksheets(1)
   
   ' Write Cell value for Q.
   objSheet.Cells(10,3).Value = SmartTags("QarsHars_QarsHars{0}")
   objSheet.Cells(11,3).Value = SmartTags("QarsHars_QarsHars{1}")
   objSheet.Cells(12,3).Value = SmartTags("QarsHars_QarsHars{2}")
   objSheet.Cells(13,3).Value = SmartTags("QarsHars_QarsHars{3}")
   objSheet.Cells(14,3).Value = SmartTags("QarsHars_QarsHars{4}")
   objSheet.Cells(16,3).Value = SmartTags("QarsHars_QarsHars{5}")
   objSheet.Cells(17,3).Value = SmartTags("QarsHars_QarsHars{0}(1)")
   objSheet.Cells(18,3).Value = SmartTags("QarsHars_QarsHars{1}(1)")
   objSheet.Cells(19,3).Value = SmartTags("QarsHars_QarsHars{2}(1)")
   objSheet.Cells(20,3).Value = SmartTags("QarsHars_QarsHars{3}(1)")
   objSheet.Cells(21,3).Value = SmartTags("QarsHars_QarsHars{4}(1)")
   objSheet.Cells(22,3).Value = SmartTags("QarsHars_QarsHars{5}(1)")
   
   ' Write Cell value for H.
   objSheet.Cells(10,4).Value = SmartTags("QarsHars_QarsHars{6}")
   objSheet.Cells(11,4).Value = SmartTags("QarsHars_QarsHars{7}")
   objSheet.Cells(12,4).Value = SmartTags("QarsHars_QarsHars{8}")
   objSheet.Cells(13,4).Value = SmartTags("QarsHars_QarsHars{9}")
   objSheet.Cells(14,4).Value = SmartTags("QarsHars_QarsHars{10}")
   objSheet.Cells(16,4).Value = SmartTags("QarsHars_QarsHars{11}")
   objSheet.Cells(17,4).Value = SmartTags("QarsHars_QarsHars{6}(1)")
   objSheet.Cells(18,4).Value = SmartTags("QarsHars_QarsHars{7}(1)")
   objSheet.Cells(19,4).Value = SmartTags("QarsHars_QarsHars{8}(1)")
   objSheet.Cells(20,4).Value = SmartTags("QarsHars_QarsHars{9}(1)")
   objSheet.Cells(21,4).Value = SmartTags("QarsHars_QarsHars{10}(1)")
   objSheet.Cells(22,4).Value = SmartTags("QarsHars_QarsHars{11}(1)")
   
   ' Write Cell value for P.
   objSheet.Cells(10,5).Value = SmartTags("shftP.Pars_shaftP{6}")
   objSheet.Cells(11,5).Value = SmartTags("shftP.Pars_shaftP{7}")
   objSheet.Cells(12,5).Value = SmartTags("shftP.Pars_shaftP{8}")
   objSheet.Cells(13,5).Value = SmartTags("shftP.Pars_shaftP{9}")
   objSheet.Cells(14,5).Value = SmartTags("shftP.Pars_shaftP{10}")
   objSheet.Cells(16,5).Value = SmartTags("shftP.Pars_shaftP{11}")
   objSheet.Cells(17,5).Value = SmartTags("shftP.Pars_shaftP{6}(1)")
   objSheet.Cells(18,5).Value = SmartTags("shftP.Pars_shaftP{7}(1)")
   objSheet.Cells(19,5).Value = SmartTags("shftP.Pars_shaftP{8}(1)")
   objSheet.Cells(20,5).Value = SmartTags("shftP.Pars_shaftP{9}(1)")
   objSheet.Cells(21,5).Value = SmartTags("shftP.Pars_shaftP{10}(1)")
   objSheet.Cells(22,5).Value = SmartTags("shftP.Pars_shaftP{11}(1)")
   
   ' Write Cell value for EFF.
   objSheet.Cells(10,6).Value = SmartTags("EFF.NPSH_EFF.NPSH{0}")
   objSheet.Cells(11,6).Value = SmartTags("EFF.NPSH_EFF.NPSH{1}")
   objSheet.Cells(12,6).Value = SmartTags("EFF.NPSH_EFF.NPSH{2}")
   objSheet.Cells(13,6).Value = SmartTags("EFF.NPSH_EFF.NPSH{3}")
   objSheet.Cells(14,6).Value = SmartTags("EFF.NPSH_EFF.NPSH{4}")
   objSheet.Cells(16,6).Value = SmartTags("EFF.NPSH_EFF.NPSH{5}")
   objSheet.Cells(17,6).Value = SmartTags("EFF.NPSH_EFF.NPSH{0}(1)")
   objSheet.Cells(18,6).Value = SmartTags("EFF.NPSH_EFF.NPSH{1}(1)")
   objSheet.Cells(19,6).Value = SmartTags("EFF.NPSH_EFF.NPSH{2}(1)")
   objSheet.Cells(20,6).Value = SmartTags("EFF.NPSH_EFF.NPSH{3}(1)")
   objSheet.Cells(21,6).Value = SmartTags("EFF.NPSH_EFF.NPSH{4}(1)")
   objSheet.Cells(22,6).Value = SmartTags("EFF.NPSH_EFF.NPSH{5}(1)")
   
   ' Save and quit.
   'objExcel.ActiveWorkbook.Save
   objExcel.ActiveWorkbook.SaveAs strSaveAsPath
   objExcel.ActiveWorkbook.Close
   objExcel.Application.Quit
   
   ' SaveAs, Print and quit.
   
   objExcel.Workbooks.Open strSaveAsPath
   objExcel.ActiveWorkbook.PrintOut
   objExcel.ActiveWorkbook.Close
*)